// TwinCAT 3 PLC project Motors
// libraries:
//   Tc2_MC2, * (Beckhoff Automation GmbH)
//   Tc2_NC, * (Beckhoff Automation GmbH)
//   Tc2_Standard, * (Beckhoff Automation GmbH)
//   Tc2_System, * (Beckhoff Automation GmbH)
//   Tc3_Module, * (Beckhoff Automation GmbH)
// project tree:
//   Data types/ TComplexStruct.TcDUT, TSimpleStruct.TcDUT
//   Global Variables/ GVL_Axis1Ctrl.TcGVL, GVL_Axis2Ctrl.TcGVL, GVL_Axis3Ctrl.TcGVL, GVL_Axis4Ctrl.TcGVL, GVL_Axis5Ctrl.TcGVL, GVL_Axis6Ctrl.TcGVL, GVL_Brakes.TcGVL, GVL_NC.TcGVL, GVL_Remote.TcGVL
//   / GlobalTextList.TcGTLO, Standard.TcTTO, Visualization Manager.TcVMO (not stored)
//   POUs/ MAIN.TcPOU, POU_AbortMoves.TcPOU, POU_AxesError.TcPOU, POU_ClearAxesErrors.TcPOU, POU_Limits.TcPOU, POU_AxisMoveAbs.TcPOU, POU_Lights.TcPOU, POU_AxisClearError.TcPOU, POU_GetPosition.TcPOU, POUNCPowerOn.TcPOU, POU_AxisJogCtrl.TcPOU, POU_SetStatus.TcPOU
//   Visualizations/ Visualization.TcVIS
// real-time tasks:
//   TASK Motors: cycle T#10ms, priority 20, ADS port 350
// motion (NC):
//   TASK NC-Task 1 SAF: cycle T#2ms, priority 4, ADS port 501
//   TASK NC-Task 1 SVB: cycle T#10ms, priority 8, ADS port 511
//   AXIS Axis 1 (id 1)
//     Dynamic: AccelerationMaximum=50, DecelerationMaximum=50, Acceleration=0.5, Deceleration=0.5, Jerk=100
//     Velo: RefSearch=5, RefSync=5, SlowManual=0.5, FastManual=3, Fast=20, Maximum=20
//     PositionAreaControl: Range=0.00025
//     TargetPosControl: Range=0.00025, Time=0.5
//     OtherSettings: AllowMotionCmdToSlave=true, PulseDistancePos=0.5, PulseDistanceNeg=0.5
//     encoder EncType=29
//       EncPara: ScaleFactorNumerator=5e-05, Offset=-200, MaxCount=#xffffffff, ReferenceSystem=1
//         SoftEndMinControl: Enable=true, Range=-169
//         SoftEndMaxControl: Enable=true, Range=175
//         Inc: RefSoftSyncMask=#x0000ffff
//     drive DrvType=24
//       DrvPara: Inverse=true
//         Analog: VeloReferenz=15, VeloScale=0.5, ScaleFactorActTorque=0.1, AccOutputDelay=0.1
//         TimeComp: TaskDelayCycles=1
//     controller CtrType=3
//       CtrPara: PriorControlFactor=1
//         PosDiffControl: Range=1
//         PID: PosKp=5, DeadBandPosition=0.0002
//         Observer: BandWidth=20
//   AXIS Axis 2 (id 2)
//     Dynamic: AccelerationMaximum=50, DecelerationMaximum=50, Acceleration=1, Deceleration=1, Jerk=0.5
//     Velo: SlowManual=0.5, FastManual=5, Maximum=10
//     PositionAreaControl: Range=0.00025
//     TargetPosControl: Range=0.00025, Time=0.5
//     OtherSettings: AllowMotionCmdToSlave=true
//     encoder EncType=29
//       EncPara: ScaleFactorNumerator=5e-05, Offset=-130, MaxCount=#xffffffff, ReferenceSystem=1
//         SoftEndMinControl: Enable=true, Range=-71
//         SoftEndMaxControl: Enable=true, Range=69
//         Inc: RefSoftSyncMask=#x0000ffff
//     drive DrvType=24
//       DrvPara: Inverse=true
//         Analog: VeloReferenz=10, ScaleFactorActTorque=0.1
//         TimeComp: TaskDelayCycles=1
//     controller CtrType=3
//       CtrPara: PriorControlFactor=1
//         PosDiffControl: Range=1
//         PID: PosKp=100, DeadBandPosition=0.0002
//         Observer: BandWidth=20
//   AXIS Axis 3 (id 3)
//     Dynamic: AccelerationMaximum=50, DecelerationMaximum=50, Acceleration=0.5, Deceleration=0.5, Jerk=100
//     Velo: RefSearch=5, RefSync=5, SlowManual=0.5, FastManual=3, Maximum=20
//     PositionAreaControl: Range=0.00025
//     TargetPosControl: Range=0.00025, Time=0.5
//     OtherSettings: AllowMotionCmdToSlave=true
//     encoder EncType=29
//       EncPara: ScaleFactorNumerator=5e-05, Offset=-200, MaxCount=#xffffffff, ReferenceSystem=1
//         SoftEndMinControl: Enable=true, Range=-169
//         SoftEndMaxControl: Enable=true, Range=175
//         Inc: RefSoftSyncMask=#x0000ffff
//     drive DrvType=24
//       DrvPara: Inverse=true
//         Analog: VeloReferenz=15, ScaleFactorActTorque=0.1
//         TimeComp: TaskDelayCycles=1
//     controller CtrType=3
//       CtrPara: PriorControlFactor=1
//         PosDiffControl: Range=1
//         PID: PosKp=5
//         Observer: BandWidth=20
//   AXIS Axis 4 (id 4)
//     Dynamic: AccelerationMaximum=50, DecelerationMaximum=50, Acceleration=0.5, Deceleration=0.5, Jerk=0.5
//     Velo: RefSearch=5, RefSync=5, SlowManual=0.5, FastManual=3, Maximum=10
//     PositionAreaControl: Range=0.00025
//     TargetPosControl: Range=0.00025
//     OtherSettings: AllowMotionCmdToSlave=true
//     encoder EncType=29
//       EncPara: ScaleFactorNumerator=5e-05, Offset=-100, MaxCount=#xffffffff, ReferenceSystem=1
//         SoftEndMinControl: Enable=true, Range=-75
//         SoftEndMaxControl: Enable=true, Range=69
//         Inc: RefSoftSyncMask=#x0000ffff
//     drive DrvType=24
//       DrvPara: Inverse=true
//         Analog: VeloReferenz=10, ScaleFactorActTorque=0.1
//         TimeComp: TaskDelayCycles=1
//     controller CtrType=3
//       CtrPara: PriorControlFactor=1
//         PosDiffControl: Range=1
//         PID: PosKp=5, DeadBandPosition=0.0002
//         Observer: BandWidth=20
//   AXIS Axis 5 (id 5)
//     Dynamic: AccelerationMaximum=50, DecelerationMaximum=50, Acceleration=0.5, Deceleration=0.5, Jerk=100
//     Velo: RefSearch=5, RefSync=5, SlowManual=0.5, FastManual=3, Maximum=20
//     PositionAreaControl: Range=0.00025
//     TargetPosControl: Range=0.00025
//     OtherSettings: AllowMotionCmdToSlave=true
//     encoder EncType=29
//       EncPara: ScaleFactorNumerator=5e-05, Offset=-200, MaxCount=#xffffffff, ReferenceSystem=1
//         SoftEndMinControl: Enable=true, Range=-169
//         SoftEndMaxControl: Enable=true, Range=175
//         Inc: RefSoftSyncMask=#x0000ffff
//     drive DrvType=24
//       DrvPara: Inverse=true
//         Analog: VeloReferenz=15, ScaleFactorActTorque=0.1
//         TimeComp: TaskDelayCycles=1
//     controller CtrType=3
//       CtrPara: PriorControlFactor=1
//         PosDiffControl: Range=1
//         PID: PosKp=5
//         Observer: BandWidth=20
//   AXIS Axis 6 (id 6)
//     Dynamic: AccelerationMaximum=50, DecelerationMaximum=50, Acceleration=0.5, Deceleration=0.5, Jerk=0.5
//     Velo: RefSearch=5, RefSync=3, SlowManual=0.5, FastManual=3, Maximum=10
//     PositionAreaControl: Range=0.00025
//     TargetPosControl: Range=0.00025
//     OtherSettings: AllowMotionCmdToSlave=true
//     encoder EncType=29
//       EncPara: ScaleFactorNumerator=5e-05, Offset=-130, MaxCount=#xffffffff, ReferenceSystem=1
//         SoftEndMinControl: Enable=true, Range=-72
//         SoftEndMaxControl: Enable=true, Range=69
//         Inc: RefSoftSyncMask=#x0000ffff
//     drive DrvType=24
//       DrvPara: Inverse=true
//         Analog: VeloReferenz=10, ScaleFactorActTorque=0.1
//         TimeComp: TaskDelayCycles=1
//     controller CtrType=3
//       CtrPara: PriorControlFactor=1
//         PosDiffControl: Range=1
//         PID: PosKp=5, DeadBandPosition=0.0002
//         Observer: BandWidth=20
// I/O:
//   DEVICE Device 1 (EtherCAT), AmsNetId 5.68.208.232.2.1
//     Term 1 (EK1200) [EK1200-5000 EtherCAT Power supply (2A E-Bus)]
//       Term 2 (EL2008) [EL2008 8Ch. Dig. Output 24V, 0.5A]
//       Term 3 (EL9011) [EL9011 End Terminal]
//   DEVICE Device 4 (EtherCAT), AmsNetId 5.68.208.232.5.1
//     Term 4 (EK1914) [EK1914, 2 Ch. Safety Input/Output 24V,  TwinSAFE]
//       modules: Module 1 (FSOE), Module 2 (DIO)
//       Term 17 (EL9410) [EL9410 E-Bus Power Supplier  (Diagnostics)]
//       Term 5 (EL5042) [EL5042 2Ch. BiSS-C Encoder]
//       Term 6 (EL5042) [EL5042 2Ch. BiSS-C Encoder]
//       Term 7 (EL5042) [EL5042 2Ch. BiSS-C Encoder]
//       Term 8 (EL7041-0052) [EL7041-0052 1Ch. Stepper motor output stage (50V, 5A)]
//       Term 9 (EL7041-0052) [EL7041-0052 1Ch. Stepper motor output stage (50V, 5A)]
//       Term 10 (EL7041-0052) [EL7041-0052 1Ch. Stepper motor output stage (50V, 5A)]
//       Term 11 (EL7041-0052) [EL7041-0052 1Ch. Stepper motor output stage (50V, 5A)]
//       Term 12 (EL7041-0052) [EL7041-0052 1Ch. Stepper motor output stage (50V, 5A)]
//       Term 13 (EL7041-0052) [EL7041-0052 1Ch. Stepper motor output stage (50V, 5A)]
//       Term 11 (EL9011) [EL9011 End Terminal]
//   DEVICE Device 3 (RT-Ethernet Protocol) (disabled), AmsNetId 5.68.208.232.4.1
//   DEVICE Device 2 (USB) (disabled)
//     Box 1 (CX2100 Power Supply)
//   DEVICE Device 5 (NOV-DP-RAM) (disabled)
// variable links:
//   NC-Task 1 SAF/Axes/Axis 1 <-> Device 4 (EtherCAT)/Term 4 (EK1914)/Term 5 (EL5042)
//     Enc/Inputs/In/nComState @bit 1 <-> WcState/InputToggle
//     Enc/Inputs/In/nComState <-> WcState/WcState
//     Enc/Inputs/In/nDataIn1 <-> FB Inputs Channel 1/Position
//     Enc/Inputs/In/nState1 @bit 12 <-> FB Inputs Channel 1/Diag
//     Enc/Inputs/In/nState1 @bit 1 <-> FB Inputs Channel 1/Error
//     Enc/Inputs/In/nState1 @bit 14 <-> FB Inputs Channel 1/Input cycle counter
//     Enc/Inputs/In/nState1 @bit 2 <-> FB Inputs Channel 1/Ready
//     Enc/Inputs/In/nState1 @bit 13 <-> FB Inputs Channel 1/TxPDO State
//     Enc/Inputs/In/nState1 <-> FB Inputs Channel 1/Warning
//   NC-Task 1 SAF/Axes/Axis 1 <-> Device 4 (EtherCAT)/Term 4 (EK1914)/Term 8 (EL7041-0052)
//     Drive/Inputs/In/nState1 @bit 3 <-> STM Status/Error
//     Drive/Inputs/In/nState1 @bit 5 <-> STM Status/Moving negative
//     Drive/Inputs/In/nState1 @bit 4 <-> STM Status/Moving positive
//     Drive/Inputs/In/nState1 @bit 1 <-> STM Status/Ready
//     Drive/Inputs/In/nState1 <-> STM Status/Ready to enable
//     Drive/Inputs/In/nState1 @bit 6 <-> STM Status/Torque reduced
//     Drive/Inputs/In/nState1 @bit 2 <-> STM Status/Warning
//     Drive/Inputs/In/nState2 @bit 3 <-> STM Status/Digital input 1
//     Drive/Inputs/In/nState2 @bit 4 <-> STM Status/Digital input 2
//     Drive/Inputs/In/nState2 @bit 5 <-> STM Status/Sync error
//     Drive/Inputs/In/nState2 @bit 7 <-> STM Status/TxPDO Toggle
//     Drive/Inputs/In/nState4 @bit 1 <-> WcState/InputToggle
//     Drive/Inputs/In/nState4 <-> WcState/WcState
//     Drive/Outputs/Out/nCtrl1 <-> STM Control/Enable
//     Drive/Outputs/Out/nCtrl1 @bit 2 <-> STM Control/Reduce torque
//     Drive/Outputs/Out/nCtrl1 @bit 1 <-> STM Control/Reset
//     Drive/Outputs/Out/nDataOut2[0] <-> STM Velocity/Velocity
//   NC-Task 1 SAF/Axes/Axis 2 <-> Device 4 (EtherCAT)/Term 4 (EK1914)/Term 5 (EL5042)
//     Enc/Inputs/In/nComState @bit 1 <-> WcState/InputToggle
//     Enc/Inputs/In/nComState <-> WcState/WcState
//     Enc/Inputs/In/nDataIn1 <-> FB Inputs Channel 2/Position
//     Enc/Inputs/In/nState1 @bit 12 <-> FB Inputs Channel 2/Diag
//     Enc/Inputs/In/nState1 @bit 1 <-> FB Inputs Channel 2/Error
//     Enc/Inputs/In/nState1 @bit 14 <-> FB Inputs Channel 2/Input cycle counter
//     Enc/Inputs/In/nState1 @bit 2 <-> FB Inputs Channel 2/Ready
//     Enc/Inputs/In/nState1 @bit 13 <-> FB Inputs Channel 2/TxPDO State
//     Enc/Inputs/In/nState1 <-> FB Inputs Channel 2/Warning
//   NC-Task 1 SAF/Axes/Axis 2 <-> Device 4 (EtherCAT)/Term 4 (EK1914)/Term 9 (EL7041-0052)
//     Drive/Inputs/In/nState1 @bit 3 <-> STM Status/Status/Error
//     Drive/Inputs/In/nState1 @bit 5 <-> STM Status/Status/Moving negative
//     Drive/Inputs/In/nState1 @bit 4 <-> STM Status/Status/Moving positive
//     Drive/Inputs/In/nState1 @bit 1 <-> STM Status/Status/Ready
//     Drive/Inputs/In/nState1 <-> STM Status/Status/Ready to enable
//     Drive/Inputs/In/nState1 @bit 6 <-> STM Status/Status/Torque reduced
//     Drive/Inputs/In/nState1 @bit 2 <-> STM Status/Status/Warning
//     Drive/Inputs/In/nState2 @bit 5 <-> STM Status/Status/Sync error
//     Drive/Inputs/In/nState2 @bit 7 <-> STM Status/Status/TxPDO Toggle
//     Drive/Inputs/In/nState4 @bit 1 <-> WcState/InputToggle
//     Drive/Inputs/In/nState4 <-> WcState/WcState
//     Drive/Outputs/Out/nCtrl1 <-> STM Control/Control/Enable
//     Drive/Outputs/Out/nCtrl1 @bit 2 <-> STM Control/Control/Reduce torque
//     Drive/Outputs/Out/nCtrl1 @bit 1 <-> STM Control/Control/Reset
//     Drive/Outputs/Out/nDataOut2[0] <-> STM Velocity/Velocity
//   NC-Task 1 SAF/Axes/Axis 3 <-> Device 4 (EtherCAT)/Term 4 (EK1914)/Term 10 (EL7041-0052)
//     Drive/Inputs/In/nState1 @bit 3 <-> STM Status/Status/Error
//     Drive/Inputs/In/nState1 @bit 5 <-> STM Status/Status/Moving negative
//     Drive/Inputs/In/nState1 @bit 4 <-> STM Status/Status/Moving positive
//     Drive/Inputs/In/nState1 @bit 1 <-> STM Status/Status/Ready
//     Drive/Inputs/In/nState1 <-> STM Status/Status/Ready to enable
//     Drive/Inputs/In/nState1 @bit 6 <-> STM Status/Status/Torque reduced
//     Drive/Inputs/In/nState1 @bit 2 <-> STM Status/Status/Warning
//     Drive/Inputs/In/nState2 @bit 5 <-> STM Status/Status/Sync error
//     Drive/Inputs/In/nState2 @bit 7 <-> STM Status/Status/TxPDO Toggle
//     Drive/Inputs/In/nState4 @bit 1 <-> WcState/InputToggle
//     Drive/Inputs/In/nState4 <-> WcState/WcState
//     Drive/Outputs/Out/nCtrl1 <-> STM Control/Control/Enable
//     Drive/Outputs/Out/nCtrl1 @bit 2 <-> STM Control/Control/Reduce torque
//     Drive/Outputs/Out/nCtrl1 @bit 1 <-> STM Control/Control/Reset
//     Drive/Outputs/Out/nDataOut2[0] <-> STM Velocity/Velocity
//   NC-Task 1 SAF/Axes/Axis 3 <-> Device 4 (EtherCAT)/Term 4 (EK1914)/Term 6 (EL5042)
//     Enc/Inputs/In/nComState @bit 1 <-> WcState/InputToggle
//     Enc/Inputs/In/nComState <-> WcState/WcState
//     Enc/Inputs/In/nDataIn1 <-> FB Inputs Channel 1/Position
//     Enc/Inputs/In/nState1 @bit 12 <-> FB Inputs Channel 1/Status/Diag
//     Enc/Inputs/In/nState1 @bit 1 <-> FB Inputs Channel 1/Status/Error
//     Enc/Inputs/In/nState1 @bit 14 <-> FB Inputs Channel 1/Status/Input cycle counter
//     Enc/Inputs/In/nState1 @bit 2 <-> FB Inputs Channel 1/Status/Ready
//     Enc/Inputs/In/nState1 @bit 13 <-> FB Inputs Channel 1/Status/TxPDO State
//     Enc/Inputs/In/nState1 <-> FB Inputs Channel 1/Status/Warning
//   NC-Task 1 SAF/Axes/Axis 4 <-> Device 4 (EtherCAT)/Term 4 (EK1914)/Term 11 (EL7041-0052)
//     Drive/Inputs/In/nState1 @bit 3 <-> STM Status/Status/Error
//     Drive/Inputs/In/nState1 @bit 5 <-> STM Status/Status/Moving negative
//     Drive/Inputs/In/nState1 @bit 4 <-> STM Status/Status/Moving positive
//     Drive/Inputs/In/nState1 @bit 1 <-> STM Status/Status/Ready
//     Drive/Inputs/In/nState1 <-> STM Status/Status/Ready to enable
//     Drive/Inputs/In/nState1 @bit 6 <-> STM Status/Status/Torque reduced
//     Drive/Inputs/In/nState1 @bit 2 <-> STM Status/Status/Warning
//     Drive/Inputs/In/nState2 @bit 5 <-> STM Status/Status/Sync error
//     Drive/Inputs/In/nState2 @bit 7 <-> STM Status/Status/TxPDO Toggle
//     Drive/Inputs/In/nState4 @bit 1 <-> WcState/InputToggle
//     Drive/Inputs/In/nState4 <-> WcState/WcState
//     Drive/Outputs/Out/nCtrl1 <-> STM Control/Control/Enable
//     Drive/Outputs/Out/nCtrl1 @bit 2 <-> STM Control/Control/Reduce torque
//     Drive/Outputs/Out/nCtrl1 @bit 1 <-> STM Control/Control/Reset
//     Drive/Outputs/Out/nDataOut2[0] <-> STM Velocity/Velocity
//   NC-Task 1 SAF/Axes/Axis 4 <-> Device 4 (EtherCAT)/Term 4 (EK1914)/Term 6 (EL5042)
//     Enc/Inputs/In/nComState @bit 1 <-> WcState/InputToggle
//     Enc/Inputs/In/nComState <-> WcState/WcState
//     Enc/Inputs/In/nDataIn1 <-> FB Inputs Channel 2/Position
//     Enc/Inputs/In/nState1 @bit 12 <-> FB Inputs Channel 2/Status/Diag
//     Enc/Inputs/In/nState1 @bit 1 <-> FB Inputs Channel 2/Status/Error
//     Enc/Inputs/In/nState1 @bit 14 <-> FB Inputs Channel 2/Status/Input cycle counter
//     Enc/Inputs/In/nState1 @bit 2 <-> FB Inputs Channel 2/Status/Ready
//     Enc/Inputs/In/nState1 @bit 13 <-> FB Inputs Channel 2/Status/TxPDO State
//     Enc/Inputs/In/nState1 <-> FB Inputs Channel 2/Status/Warning
//   NC-Task 1 SAF/Axes/Axis 5 <-> Device 4 (EtherCAT)/Term 4 (EK1914)/Term 12 (EL7041-0052)
//     Drive/Inputs/In/nState1 @bit 3 <-> STM Status/Status/Error
//     Drive/Inputs/In/nState1 @bit 5 <-> STM Status/Status/Moving negative
//     Drive/Inputs/In/nState1 @bit 4 <-> STM Status/Status/Moving positive
//     Drive/Inputs/In/nState1 @bit 1 <-> STM Status/Status/Ready
//     Drive/Inputs/In/nState1 <-> STM Status/Status/Ready to enable
//     Drive/Inputs/In/nState1 @bit 6 <-> STM Status/Status/Torque reduced
//     Drive/Inputs/In/nState1 @bit 2 <-> STM Status/Status/Warning
//     Drive/Inputs/In/nState2 @bit 3 <-> STM Status/Status/Digital input 1
//     Drive/Inputs/In/nState2 @bit 4 <-> STM Status/Status/Digital input 2
//     Drive/Inputs/In/nState2 @bit 5 <-> STM Status/Status/Sync error
//     Drive/Inputs/In/nState2 @bit 7 <-> STM Status/Status/TxPDO Toggle
//     Drive/Inputs/In/nState4 @bit 1 <-> WcState/InputToggle
//     Drive/Inputs/In/nState4 <-> WcState/WcState
//     Drive/Outputs/Out/nCtrl1 <-> STM Control/Control/Enable
//     Drive/Outputs/Out/nCtrl1 @bit 2 <-> STM Control/Control/Reduce torque
//     Drive/Outputs/Out/nCtrl1 @bit 1 <-> STM Control/Control/Reset
//     Drive/Outputs/Out/nDataOut2[0] <-> STM Velocity/Velocity
//   NC-Task 1 SAF/Axes/Axis 5 <-> Device 4 (EtherCAT)/Term 4 (EK1914)/Term 7 (EL5042)
//     Enc/Inputs/In/nComState @bit 1 <-> WcState/InputToggle
//     Enc/Inputs/In/nComState <-> WcState/WcState
//     Enc/Inputs/In/nDataIn1 <-> FB Inputs Channel 1/Position
//     Enc/Inputs/In/nState1 @bit 12 <-> FB Inputs Channel 1/Status/Diag
//     Enc/Inputs/In/nState1 @bit 1 <-> FB Inputs Channel 1/Status/Error
//     Enc/Inputs/In/nState1 @bit 14 <-> FB Inputs Channel 1/Status/Input cycle counter
//     Enc/Inputs/In/nState1 @bit 2 <-> FB Inputs Channel 1/Status/Ready
//     Enc/Inputs/In/nState1 @bit 13 <-> FB Inputs Channel 1/Status/TxPDO State
//     Enc/Inputs/In/nState1 <-> FB Inputs Channel 1/Status/Warning
//   NC-Task 1 SAF/Axes/Axis 6 <-> Device 4 (EtherCAT)/Term 4 (EK1914)/Term 13 (EL7041-0052)
//     Drive/Inputs/In/nState1 @bit 3 <-> STM Status/Status/Error
//     Drive/Inputs/In/nState1 @bit 5 <-> STM Status/Status/Moving negative
//     Drive/Inputs/In/nState1 @bit 4 <-> STM Status/Status/Moving positive
//     Drive/Inputs/In/nState1 @bit 1 <-> STM Status/Status/Ready
//     Drive/Inputs/In/nState1 <-> STM Status/Status/Ready to enable
//     Drive/Inputs/In/nState1 @bit 6 <-> STM Status/Status/Torque reduced
//     Drive/Inputs/In/nState1 @bit 2 <-> STM Status/Status/Warning
//     Drive/Inputs/In/nState2 @bit 5 <-> STM Status/Status/Sync error
//     Drive/Inputs/In/nState2 @bit 7 <-> STM Status/Status/TxPDO Toggle
//     Drive/Inputs/In/nState4 @bit 1 <-> WcState/InputToggle
//     Drive/Inputs/In/nState4 <-> WcState/WcState
//     Drive/Outputs/Out/nCtrl1 <-> STM Control/Control/Enable
//     Drive/Outputs/Out/nCtrl1 @bit 2 <-> STM Control/Control/Reduce torque
//     Drive/Outputs/Out/nCtrl1 @bit 1 <-> STM Control/Control/Reset
//     Drive/Outputs/Out/nDataOut2[0] <-> STM Velocity/Velocity
//   NC-Task 1 SAF/Axes/Axis 6 <-> Device 4 (EtherCAT)/Term 4 (EK1914)/Term 7 (EL5042)
//     Enc/Inputs/In/nComState @bit 1 <-> WcState/InputToggle
//     Enc/Inputs/In/nComState <-> WcState/WcState
//     Enc/Inputs/In/nDataIn1 <-> FB Inputs Channel 2/Position
//     Enc/Inputs/In/nState1 @bit 12 <-> FB Inputs Channel 2/Status/Diag
//     Enc/Inputs/In/nState1 @bit 1 <-> FB Inputs Channel 2/Status/Error
//     Enc/Inputs/In/nState1 @bit 14 <-> FB Inputs Channel 2/Status/Input cycle counter
//     Enc/Inputs/In/nState1 @bit 2 <-> FB Inputs Channel 2/Status/Ready
//     Enc/Inputs/In/nState1 @bit 13 <-> FB Inputs Channel 2/Status/TxPDO State
//     Enc/Inputs/In/nState1 <-> FB Inputs Channel 2/Status/Warning
//   Motors/Motors Instance <-> Device 1 (EtherCAT)/Term 1 (EK1200)/Term 2 (EL2008)
//     Standard Outputs/MAIN.bAxis{1..6}Brake <-> Channel {1..6}/Output  (6 links)
//   Motors/Motors Instance <-> Device 4 (EtherCAT)/Term 4 (EK1914)
//     Standard Inputs/MAIN.bESTOP <-> Module 2 (DIO)/DIO Inputs/Input 0
//     Standard Outputs/POU_Lights.bLightAmber <-> Module 2 (DIO)/DIO Outputs/Output 1
//     Standard Outputs/POU_Lights.bLightGreen <-> Module 2 (DIO)/DIO Outputs/Output 0
//     Standard Outputs/POU_Lights.bLightRed <-> Module 2 (DIO)/DIO Outputs/Output 2
//   Motors/Motors Instance <-> Device 4 (EtherCAT)/Term 4 (EK1914)/Term 10 (EL7041-0052)
//     Standard Inputs/POUNCPowerOn.bAxis3LimitNegI <-> STM Status/Status/Digital input 2
//     Standard Inputs/POUNCPowerOn.bAxis3LimitPosI <-> STM Status/Status/Digital input 1
//     Standard Inputs/POU_Limits.bAxis3LimitNegI <-> STM Status/Status/Digital input 2
//     Standard Inputs/POU_Limits.bAxis3LimitPosI <-> STM Status/Status/Digital input 1
//   Motors/Motors Instance <-> Device 4 (EtherCAT)/Term 4 (EK1914)/Term 11 (EL7041-0052)
//     Standard Inputs/POUNCPowerOn.bAxis4LimitNegI <-> STM Status/Status/Digital input 2
//     Standard Inputs/POUNCPowerOn.bAxis4LimitPosI <-> STM Status/Status/Digital input 1
//     Standard Inputs/POU_Limits.bAxis4LimitNegI <-> STM Status/Status/Digital input 2
//     Standard Inputs/POU_Limits.bAxis4LimitPosI <-> STM Status/Status/Digital input 1
//   Motors/Motors Instance <-> Device 4 (EtherCAT)/Term 4 (EK1914)/Term 12 (EL7041-0052)
//     Standard Inputs/POUNCPowerOn.bAxis5LimitNegI <-> STM Status/Status/Digital input 2
//     Standard Inputs/POUNCPowerOn.bAxis5LimitPosI <-> STM Status/Status/Digital input 1
//     Standard Inputs/POU_Limits.bAxis5LimitNegI <-> STM Status/Status/Digital input 2
//     Standard Inputs/POU_Limits.bAxis5LimitPosI <-> STM Status/Status/Digital input 1
//   Motors/Motors Instance <-> Device 4 (EtherCAT)/Term 4 (EK1914)/Term 13 (EL7041-0052)
//     Standard Inputs/POUNCPowerOn.bAxis6LimitNegI <-> STM Status/Status/Digital input 2
//     Standard Inputs/POUNCPowerOn.bAxis6LimitPosI <-> STM Status/Status/Digital input 1
//     Standard Inputs/POU_Limits.bAxis6LimitNegI <-> STM Status/Status/Digital input 2
//     Standard Inputs/POU_Limits.bAxis6LimitPosI <-> STM Status/Status/Digital input 1
//   Motors/Motors Instance <-> Device 4 (EtherCAT)/Term 4 (EK1914)/Term 8 (EL7041-0052)
//     Standard Inputs/POUNCPowerOn.bAxis1LimitNegI <-> STM Status/Digital input 2
//     Standard Inputs/POUNCPowerOn.bAxis1LimitPosI <-> STM Status/Digital input 1
//     Standard Inputs/POU_Limits.bAxis1LimitNegI <-> STM Status/Digital input 2
//     Standard Inputs/POU_Limits.bAxis1LimitPosI <-> STM Status/Digital input 1
//   Motors/Motors Instance <-> Device 4 (EtherCAT)/Term 4 (EK1914)/Term 9 (EL7041-0052)
//     Standard Inputs/POUNCPowerOn.bAxis2LimitNegI <-> STM Status/Status/Digital input 2
//     Standard Inputs/POUNCPowerOn.bAxis2LimitPosI <-> STM Status/Status/Digital input 1
//     Standard Inputs/POU_Limits.bAxis2LimitNegI <-> STM Status/Status/Digital input 2
//     Standard Inputs/POU_Limits.bAxis2LimitPosI <-> STM Status/Status/Digital input 1
//   Motors/Motors Instance <-> NC-Task 1 SAF/Axes/Axis 1
//     Standard Inputs/GVL_NC.Axis1.NcToPlc <-> Outputs/ToPlc
//     Standard Inputs/POU_AxesError.bAxis1ErrorI <-> Outputs/ToPlc/StateDWord/Error
//     Standard Outputs/GVL_NC.Axis1.PlcToNc <-> Inputs/FromPlc
//   Motors/Motors Instance <-> NC-Task 1 SAF/Axes/Axis 2
//     Standard Inputs/GVL_NC.Axis2.NcToPlc <-> Outputs/ToPlc
//     Standard Inputs/POU_AxesError.bAxis2ErrorI <-> Outputs/ToPlc/StateDWord/Error
//     Standard Outputs/GVL_NC.Axis2.PlcToNc <-> Inputs/FromPlc
//   Motors/Motors Instance <-> NC-Task 1 SAF/Axes/Axis 3
//     Standard Inputs/GVL_NC.Axis3.NcToPlc <-> Outputs/ToPlc
//     Standard Inputs/POU_AxesError.bAxis3ErrorI <-> Outputs/ToPlc/StateDWord/Error
//     Standard Outputs/GVL_NC.Axis3.PlcToNc <-> Inputs/FromPlc
//   Motors/Motors Instance <-> NC-Task 1 SAF/Axes/Axis 4
//     Standard Inputs/GVL_NC.Axis4.NcToPlc <-> Outputs/ToPlc
//     Standard Inputs/POU_AxesError.bAxis4ErrorI <-> Outputs/ToPlc/StateDWord/Error
//     Standard Outputs/GVL_NC.Axis4.PlcToNc <-> Inputs/FromPlc
//   Motors/Motors Instance <-> NC-Task 1 SAF/Axes/Axis 5
//     Standard Inputs/GVL_NC.Axis5.NcToPlc <-> Outputs/ToPlc
//     Standard Inputs/POU_AxesError.bAxis5ErrorI <-> Outputs/ToPlc/StateDWord/Error
//     Standard Outputs/GVL_NC.Axis5.PlcToNc <-> Inputs/FromPlc
//   Motors/Motors Instance <-> NC-Task 1 SAF/Axes/Axis 6
//     Standard Inputs/GVL_NC.Axis6.NcToPlc <-> Outputs/ToPlc
//     Standard Inputs/POU_AxesError.bAxis6ErrorI <-> Outputs/ToPlc/StateDWord/Error
//     Standard Outputs/GVL_NC.Axis6.PlcToNc <-> Inputs/FromPlc

CONFIGURATION Motors
    RESOURCE PLC ON TwinCAT3
        TASK Standard(INTERVAL := T#10ms, PRIORITY := 20);
        PROGRAM MAIN WITH Standard : MAIN;
    END_RESOURCE
END_CONFIGURATION

// ---- Data types/TComplexStruct.TcDUT
TYPE TComplexStruct :
STRUCT
	intVal : INT:=1200;
	dintArr: ARRAY[0..3] OF DINT:=[ 1,2,3,4];
	boolVal: BOOL := FALSE;
	byteVal: BYTE:=10;
	stringVal : STRING(5) := 'hallo';
	simpleStruct1: TSimpleStruct;
END_STRUCT
END_TYPE

// ---- Data types/TSimpleStruct.TcDUT
TYPE TSimpleStruct :
STRUCT
	lrealVal: LREAL := 1.23;
	dintVal1: DINT := 120000;
END_STRUCT
END_TYPE

// ---- Global Variables/GVL_Axis1Ctrl.TcGVL
VAR_GLOBAL
	bAxis1Enable:BOOL;
	bAxis1EnablePos:BOOL:=TRUE;
	bAxis1EnableNeg:BOOL:=TRUE;
	bAxis1JogPos:BOOL;
	bAxis1JogNeg:BOOL;
	rAxis1Target:LREAL;
	bAxis1MoveABS:BOOL;
	rAxis1Vel:REAL;
	bAxis1PosLimit:BOOL:=TRUE;
	bAxis1NegLimit:BOOL:=TRUE;
	bAxis1GetPos:BOOL:=FALSE;
	rAxis1Position:LREAL;
	bAxis1InPosition:BOOL;
	iAxis1Error:UDINT;
	bAxis1Error:BOOL;
	bReset1Done:BOOL:=FALSE;
	
	
	
END_VAR

// ---- Global Variables/GVL_Axis2Ctrl.TcGVL
VAR_GLOBAL
	bAxis2Enable:BOOL;
	bAxis2EnablePos:BOOL:=TRUE;
	bAxis2EnableNeg:BOOL:=TRUE;
	bAxis2JogPos:BOOL;
	bAxis2JogNeg:BOOL;
	rAxis2Target:LREAL;
	bAxis2MoveABS:BOOL;
	rAxis2Vel:REAL;
	bAxis2PosLimit:BOOL:=TRUE;
	bAxis2NegLimit:BOOL:=TRUE;
	bAxis2GetPos:BOOL:=FALSE;
	rAxis2Position:LREAL;
	bAxis2InPosition:BOOL;
	iAxis2Error:UDINT;
	bAxis2Error:BOOL;
	bReset2Done:BOOL:=FALSE;
END_VAR

// ---- Global Variables/GVL_Axis3Ctrl.TcGVL
VAR_GLOBAL
	bAxis3Enable:BOOL;
	bAxis3EnablePos:BOOL:=TRUE;
	bAxis3EnableNeg:BOOL:=TRUE;
	bAxis3JogPos:BOOL;
	bAxis3JogNeg:BOOL;
	rAxis3Target:LREAL;
	bAxis3MoveABS:BOOL;
	rAxis3Vel:REAL;
	bAxis3PosLimit:BOOL:=TRUE;
	bAxis3NegLimit:BOOL:=TRUE;
	bAxis3GetPos:BOOL:=FALSE;
	rAxis3Position:LREAL;
	bAxis3InPosition:BOOL;
	iAxis3Error:UDINT;
	bAxis3Error:BOOL;
	bReset3Done:BOOL:=FALSE;
END_VAR

// ---- Global Variables/GVL_Axis4Ctrl.TcGVL
VAR_GLOBAL
	bAxis4Enable:BOOL;
	bAxis4EnablePos:BOOL:=TRUE;
	bAxis4EnableNeg:BOOL:=TRUE;
	bAxis4JogPos:BOOL;
	bAxis4JogNeg:BOOL;
	rAxis4Target:LREAL;
	bAxis4MoveABS:BOOL;
	rAxis4Vel:REAL;
	bAxis4PosLimit:BOOL:=TRUE;
	bAxis4NegLimit:BOOL:=TRUE;
	bAxis4GetPos:BOOL:=FALSE;
	rAxis4Position:LREAL;
	bAxis4InPosition:BOOL;
	iAxis4Error:UDINT;
	bAxis4Error:BOOL;
	bReset4Done:BOOL:=FALSE;
END_VAR

// ---- Global Variables/GVL_Axis5Ctrl.TcGVL
VAR_GLOBAL
	bAxis5Enable:BOOL;
	bAxis5EnablePos:BOOL:=TRUE;
	bAxis5EnableNeg:BOOL:=TRUE;
	bAxis5JogPos:BOOL;
	bAxis5JogNeg:BOOL;
	rAxis5Target:LREAL;
	bAxis5MoveABS:BOOL;
	rAxis5Vel:REAL;
	bAxis5PosLimit:BOOL:=TRUE;
	bAxis5NegLimit:BOOL:=TRUE;
	bAxis5GetPos:BOOL:=FALSE;
	rAxis5Position:LREAL;
	bAxis5InPosition:BOOL;	
	iAxis5Error:UDINT;
	bAxis5Error:BOOL;
	bReset5Done:BOOL:=FALSE;
END_VAR

// ---- Global Variables/GVL_Axis6Ctrl.TcGVL
VAR_GLOBAL
	bAxis6Enable:BOOL;
	bAxis6EnablePos:BOOL:=TRUE;
	bAxis6EnableNeg:BOOL:=TRUE;
	bAxis6JogPos:BOOL;
	bAxis6JogNeg:BOOL;
	rAxis6Target:LREAL;
	bAxis6MoveABS:BOOL;
	rAxis6Vel:REAL;
	bAxis6PosLimit:BOOL:=TRUE;
	bAxis6NegLimit:BOOL:=TRUE;
	bAxis6GetPos:BOOL:=FALSE;
	rAxis6Position:LREAL;
	bAxis6InPosition:BOOL;
	iAxis6Error:UDINT;
	bAxis6Error:BOOL;
	bReset6Done:BOOL:=FALSE;
END_VAR

// ---- Global Variables/GVL_Brakes.TcGVL
VAR_GLOBAL
	bAxis1Brake:BOOL;
	bAxis2Brake:BOOL;
	bAxis3Brake:BOOL;
	bAxis4Brake:BOOL;
	bAxis5Brake:BOOL;
	bAxis6Brake:BOOL;
END_VAR

// ---- Global Variables/GVL_NC.TcGVL
VAR_GLOBAL
	Axis1:AXIS_REF;
	stAxis1:ST_AxisStatus;
	Axis2:AXIS_REF;
	stAxis2:ST_AxisStatus;
	Axis3:AXIS_REF;
	stAxis3:ST_AxisStatus;
	Axis4:AXIS_REF;
	stAxis4:ST_AxisStatus;	
	Axis5:AXIS_REF;
	stAxis5:ST_AxisStatus;
	Axis6:AXIS_REF;
	stAxis6:ST_AxisStatus;
	rAxisVelV:REAL:=2;
	rAxisVelH:REAL:=2;
	bLimits:BOOL;
	bMotorError:BOOL:=FALSE;
	bReSetMotor:BOOL:=FALSE;
	bAbortMove:BOOL:=FALSE;
END_VAR

// ---- Global Variables/GVL_Remote.TcGVL
VAR_GLOBAL
	bRemote:BOOL:=TRUE;
END_VAR

// ---- POUs/MAIN.TcPOU
PROGRAM MAIN
VAR
	(*primitive Types*)
	Bool1:BOOL := FALSE;
	int1:INT :=0;
	dint1:DINT:=125000;
	usint1:USINT:=200;
	real1:REAL:= 1.2;
	lreal1:LREAL:=3.5;
	rConst:REAL;
	bClearAxesErrorm:BOOL:=FALSE;
	
	bAxis1Brake  AT%Q* : BOOL;
	bAxis2Brake  AT%Q* : BOOL;
	bAxis3Brake  AT%Q* : BOOL;
	bAxis4Brake  AT%Q* : BOOL;
	bAxis5Brake  AT%Q* : BOOL;
	bAxis6Brake  AT%Q* : BOOL;
	
	
	
	(*string Types*)
	str1:STRING := 'this is a test string';
	str2:STRING(5) := 'hallo';
	
	(*struct Types*)
	complexStruct1 : TComplexStruct;

	bESTOP AT%I* :BOOL;
	i: INT;
//Axis 1 Var	
	fbReadAxis1Status:MC_ReadStatus;
	bAxesEnablem:BOOL:=FALSE;
	bAxis1JogPosm:BOOL:=FALSE;
	bAxis1JogNegm:BOOL:=FALSE;
	rAxis1Targetm:LREAL:=0;
	rAxis1Positionm:LREAL:=0;
	bAxis1LimitPos:BOOL;
	bAxis1LimitNeg:BOOL;
	bAxis1MoveABSm:BOOL:=FALSE;
	bAxis1GetPosm:BOOL:=FALSE;
	bAxis1InPositionm:BOOL;
//Axis 2 Var	
	fbReadAxis2Status:MC_ReadStatus;
	bAxis2Enablem:BOOL:=FALSE;
	bAxis2JogPosm:BOOL:=FALSE;
	bAxis2JogNegm:BOOL:=FALSE;
	rAxis2Targetm:LREAL:=0;
	rAxis2Positionm:LREAL:=0;
	bAxis2LimitPos:BOOL;
	bAxis2LimitNeg:BOOL;
	bAxis2MoveABSm:BOOL:=FALSE;
	bAxis2InPositionm:BOOL;
//Axis 3 Var	
	fbReadAxis3Status:MC_ReadStatus;	
	bAxis3Enablem:BOOL:=FALSE;
	bAxis3JogPosm:BOOL:=FALSE;
	bAxis3JogNegm:BOOL:=FALSE;
	rAxis3Targetm:LREAL:=0;
	rAxis3Positionm:LREAL:=0;
	bAxis3LimitPos:BOOL;
	bAxis3LimitNeg:BOOL;
	bAxis3MoveABSm:BOOL:=FALSE;
	bAxis3InPositionm:BOOL;
//Axis 4 Var	
	fbReadAxis4Status:MC_ReadStatus;
	bAxis4JogPosm:BOOL:=FALSE;
	bAxis4JogNegm:BOOL:=FALSE;
	rAxis4Targetm:LREAL:=0;
	rAxis4Positionm:LREAL:=0;
	bAxis4LimitPos:BOOL;
	bAxis4LimitNeg:BOOL;
	bAxis4MoveABSm:BOOL:=FALSE;
	bAxis4InPositionm:BOOL;
//Axis 5 Var	
	fbReadAxis5Status:MC_ReadStatus;
	bAxis5JogPosm:BOOL:=FALSE;
	bAxis5JogNegm:BOOL:=FALSE;
	rAxis5Targetm:LREAL:=0;
	rAxis5Positionm:LREAL:=0;
	bAxis5LimitPos:BOOL;
	bAxis5LimitNeg:BOOL;
	bAxis5MoveABSm:BOOL:=FALSE;
	bAxis5InPositionm:BOOL;
//Axis 6 Var	
	fbReadAxis6Status:MC_ReadStatus;
	bAxis6JogPosm:BOOL:=FALSE;
	bAxis6JogNegm:BOOL:=FALSE;
	rAxis6Targetm:LREAL:=0;
	rAxis6Positionm:LREAL:=0;
	bAxis6LimitPos:BOOL;
	bAxis6LimitNeg:BOOL;
	bAxis6MoveABSm:BOOL:=FALSE;
	bAxis6InPositionm:BOOL;

	fbMoveAbs: MC_MoveAbsolute;
	fbMoveAbs2: MC_MoveAbsolute;
END_VAR


	POU_GetPosition();
	POU_Lights(bEStop:=bEStop);
	POU_Limits();
	POU_AxesError();
IF bESTOP AND bLimits AND bMotorError
	THEN
	IF bRemote 
	THEN

	//Axis 1
	bAxis1Enable:=bAxesEnablem;
	bAxis1Brake:=bAxis1Enable;
	rAxis1Target:=rAxis1Targetm;
	bAxis1MoveABS:=bAxis1MoveABSm;
	rAxis1Positionm:=rAxis1Position;
	bAxis1InPositionm:=bAxis1InPosition;

	//Axis 2
	bAxis2Enable:=bAxesEnablem;
	bAxis2Brake:=bAxis2Enable;
	rAxis2Target:=rAxis2Targetm;
	bAxis2MoveABS:=bAxis2MoveABSm;
	rAxis2Positionm:=rAxis2Position;
	bAxis2InPositionm:=bAxis2InPosition;

	//Axis 3
	bAxis3Enable:=bAxesEnablem;
	bAxis3Brake:=bAxis3Enable;
	rAxis3Target:=rAxis3Targetm;
	bAxis3MoveABS:=bAxis3MoveABSm;
	rAxis3Positionm:=rAxis3Position;
	bAxis3InPositionm:=bAxis3InPosition;

	//Axis 4
	bAxis4Enable:=bAxesEnablem;
	bAxis4Brake:=bAxis4Enable;
	rAxis4Target:=rAxis4Targetm;
	bAxis4MoveABS:=bAxis4MoveABSm;
	rAxis4Positionm:=rAxis4Position;
	bAxis4InPositionm:=bAxis4InPosition;

	//Axis 5
	bAxis5Enable:=bAxesEnablem;
	bAxis5Brake:=bAxis5Enable;
	rAxis5Target:=rAxis5Targetm;
	bAxis5MoveABS:=bAxis5MoveABSm;
	rAxis5Positionm:=rAxis5Position;
	bAxis5InPositionm:=bAxis5InPosition;

	//Axis 6
	bAxis6Enable:=bAxesEnablem;
	bAxis6Brake:=bAxis6Enable;
	rAxis6Target:=rAxis6Targetm;
	bAxis6MoveABS:=bAxis6MoveABSm;
	rAxis6Positionm:=rAxis6Position;
	bAxis6InPositionm:=bAxis6InPosition;

	POUNCPowerOn();
	POU_AxisJogCtrl();
	POU_AxisMoveABS();

	END_IF;
ELSE
	bAxis1Enable:=FALSE;
	bAxis2Enable:=FALSE;
	bAxis3Enable:=FALSE;
	bAxis4Enable:=FALSE;
	bAxis5Enable:=FALSE;
	bAxis6Enable:=FALSE;
	bAxis1MoveABS:=FALSE;
	bAxis2MoveABS:=FALSE;
	bAxis3MoveABS:=FALSE;
	bAxis4MoveABS:=FALSE;
	bAxis5MoveABS:=FALSE;
	bAxis6MoveABS:=FALSE;
	bAxis1Brake:=FALSE;
	bAxis2Brake:=FALSE;
	bAxis3Brake:=FALSE;
	bAxis4Brake:=FALSE;
	bAxis5Brake:=FALSE;
	bAxis6Brake:=FALSE;
	//needs to set move abs execute to false both 1 and 2
	POUNCPowerOn();
END_IF;
IF bClearAxesErrorm
	THEN
	int1:=int1+1;
	bReSetMotor:=TRUE;
	POU_ClearAxesErrors();

	IF bReset2Done
		THEN
			bReSetMotor:=FALSE;
			POU_ClearAxesErrors();
			bClearAxesErrorm:=FALSE;
	END_IF

END_IF

END_PROGRAM

// ---- POUs/POU_GetPosition.TcPOU
PROGRAM POU_GetPosition
VAR
	fb_Axis1Position:MC_ReadActualPosition;
	fb_Axis2Position:MC_ReadActualPosition;
	fb_Axis3Position:MC_ReadActualPosition;
	fb_Axis4Position:MC_ReadActualPosition;
	fb_Axis5Position:MC_ReadActualPosition;
	fb_Axis6Position:MC_ReadActualPosition;
END_VAR

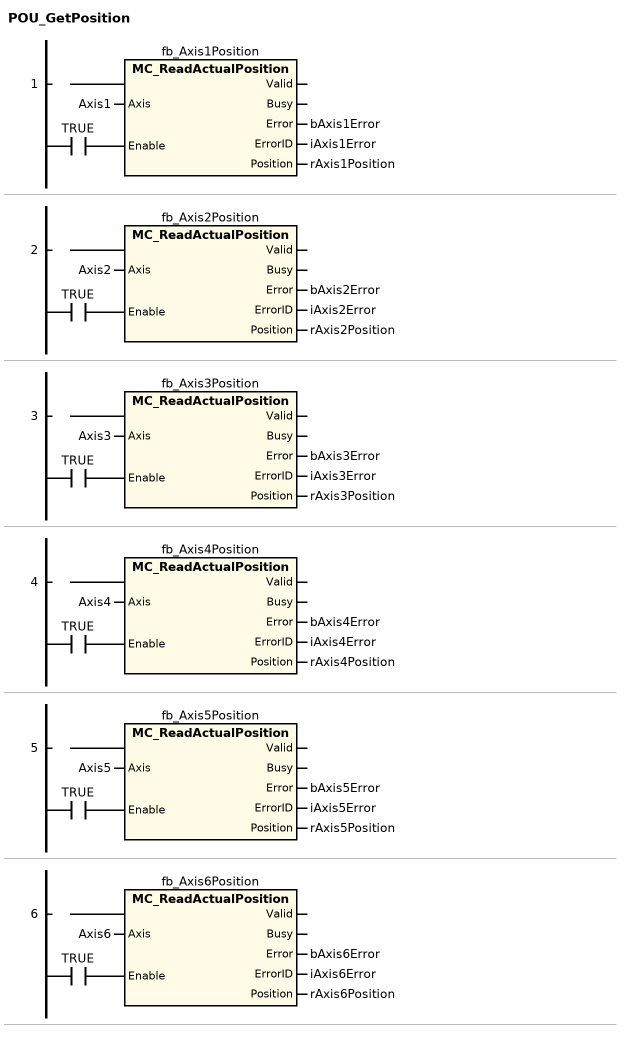
// NETWORK 1
fb_Axis1Position(
    Axis := Axis1,
    Enable := TRUE,
    Error => bAxis1Error,
    ErrorID => iAxis1Error,
    Position => rAxis1Position); // MC_ReadActualPosition

// NETWORK 2
fb_Axis2Position(
    Axis := Axis2,
    Enable := TRUE,
    Error => bAxis2Error,
    ErrorID => iAxis2Error,
    Position => rAxis2Position); // MC_ReadActualPosition

// NETWORK 3
fb_Axis3Position(
    Axis := Axis3,
    Enable := TRUE,
    Error => bAxis3Error,
    ErrorID => iAxis3Error,
    Position => rAxis3Position); // MC_ReadActualPosition

// NETWORK 4
fb_Axis4Position(
    Axis := Axis4,
    Enable := TRUE,
    Error => bAxis4Error,
    ErrorID => iAxis4Error,
    Position => rAxis4Position); // MC_ReadActualPosition

// NETWORK 5
fb_Axis5Position(
    Axis := Axis5,
    Enable := TRUE,
    Error => bAxis5Error,
    ErrorID => iAxis5Error,
    Position => rAxis5Position); // MC_ReadActualPosition

// NETWORK 6
fb_Axis6Position(
    Axis := Axis6,
    Enable := TRUE,
    Error => bAxis6Error,
    ErrorID => iAxis6Error,
    Position => rAxis6Position); // MC_ReadActualPosition

END_PROGRAM

// ---- POUs/POU_Lights.TcPOU
PROGRAM POU_Lights
VAR_INPUT
bAxesEnablem:BOOL;
bEStop:BOOL;
END_VAR
VAR
tTimeLightOn:TIME:=T#0S;
tTimeStartMove:TIME;
tCurrentLight:TIME;
tCurrentMoveDur:TIME;
bLightRed  AT%Q* : BOOL;
bLightAmber  AT%Q* : BOOL;
bLightGreen  AT%Q* : BOOL;
END_VAR

IF bEStop AND bLimits AND bMotorError
	THEN
	

IF bAxis1Enable OR bAxis2Enable OR bAxis3Enable OR bAxis4Enable OR bAxis5Enable OR bAxis6Enable
	
	THEN
	tCurrentLight:=TIME();
	tCurrentMoveDur:=tCurrentLight-tTimeLightOn;
	IF (tCurrentMoveDur < T#1S)  
		THEN
		bLightRed:=FALSE;
		bLightAmber:=TRUE;
		bLightGreen:=FALSE;
	END_IF
	IF (tCurrentMoveDur > T#1S)AND (tCurrentMoveDur < T#2S)
		THEN
		bLightRed:=FALSE;
		bLightAmber:=FALSE;
		bLightGreen:=FALSE;
	END_IF
	IF (tCurrentMoveDur > T#2S)
		THEN
		tTimeLightOn:=TIME();
	END_IF
	ELSE
	tTimeLightOn:=TIME();	
	bLightRed:=FALSE;
	bLightAmber:=FALSE;
	bLightGreen:=TRUE;
END_IF
ELSE
	bLightRed:=TRUE;
	bLightAmber:=FALSE;
	bLightGreen:=FALSE;
END_IF

END_PROGRAM

// ---- POUs/POU_Limits.TcPOU
PROGRAM POU_Limits
VAR
	bAxis1LimitPosI AT%I* :BOOL;
	bAxis1LimitNegI AT%I* :BOOL;
	bAxis2LimitPosI AT%I* :BOOL;
	bAxis2LimitNegI AT%I* :BOOL;
	bAxis3LimitPosI AT%I* :BOOL;
	bAxis3LimitNegI AT%I* :BOOL;
	bAxis4LimitPosI AT%I* :BOOL;
	bAxis4LimitNegI AT%I* :BOOL;
	bAxis5LimitPosI AT%I* :BOOL;
	bAxis5LimitNegI AT%I* :BOOL;
	bAxis6LimitPosI AT%I* :BOOL;
	bAxis6LimitNegI AT%I* :BOOL;
END_VAR

IF bAxis1LimitPosI AND bAxis1LimitNegI AND bAxis2LimitPosI AND bAxis2LimitNegI AND bAxis3LimitPosI AND bAxis3LimitNegI AND bAxis4LimitPosI AND bAxis4LimitNegI AND bAxis5LimitPosI AND bAxis5LimitNegI AND bAxis6LimitPosI AND bAxis6LimitNegI
	THEN bLimits:= TRUE;
	ELSE bLimits:=FALSE;
END_IF

END_PROGRAM

// ---- POUs/POU_AxesError.TcPOU
PROGRAM POU_AxesError
VAR
	bAxis1ErrorI AT%I* :BOOL;
	bAxis2ErrorI AT%I* :BOOL;
	bAxis3ErrorI AT%I* :BOOL;
	bAxis4ErrorI AT%I* :BOOL;
	bAxis5ErrorI AT%I* :BOOL;
	bAxis6ErrorI AT%I* :BOOL;
END_VAR

IF bAxis1ErrorI OR bAxis2ErrorI OR bAxis3ErrorI OR bAxis4ErrorI OR bAxis5ErrorI OR bAxis6ErrorI
	THEN
	bMotorError:=FALSE;
	ELSE
		bMotorError:=TRUE;
END_IF

END_PROGRAM

// ---- POUs/POUNCPowerOn.TcPOU
PROGRAM POUNCPowerOn
VAR
	fbAxis1PowerOn:MC_Power;
	fbAxis2PowerOn:MC_Power;
	fbAxis3PowerOn:MC_Power;
	fbAxis4PowerOn:MC_Power;
	fbAxis5PowerOn:MC_Power;
	fbAxis6PowerOn:MC_Power;
	bAxis1LimitPosI AT%I* :BOOL;
	bAxis1LimitNegI AT%I* :BOOL;
	bAxis2LimitPosI AT%I* :BOOL;
	bAxis2LimitNegI AT%I* :BOOL;
	bAxis3LimitPosI AT%I* :BOOL;
	bAxis3LimitNegI AT%I* :BOOL;
	bAxis4LimitPosI AT%I* :BOOL;
	bAxis4LimitNegI AT%I* :BOOL;
	bAxis5LimitPosI AT%I* :BOOL;
	bAxis5LimitNegI AT%I* :BOOL;
	bAxis6LimitPosI AT%I* :BOOL;
	bAxis6LimitNegI AT%I* :BOOL;
END_VAR

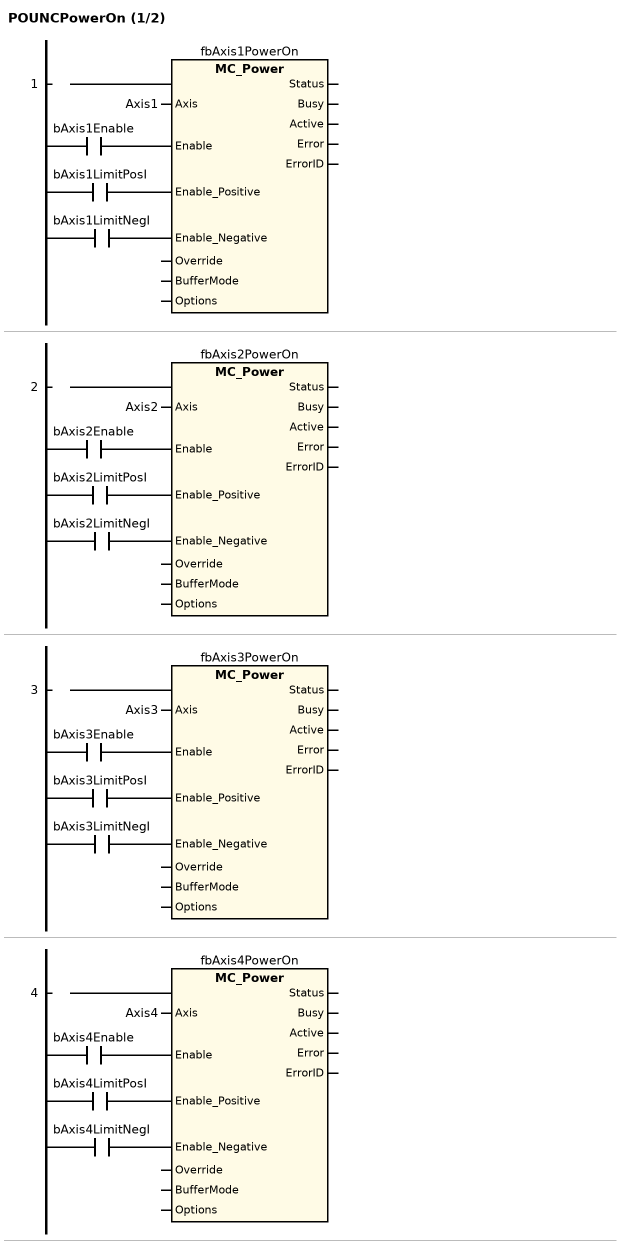
// NETWORK 1
fbAxis1PowerOn(
    Axis := Axis1,
    Enable := bAxis1Enable,
    Enable_Positive := bAxis1LimitPosI,
    Enable_Negative := bAxis1LimitNegI); // MC_Power

// NETWORK 2
fbAxis2PowerOn(
    Axis := Axis2,
    Enable := bAxis2Enable,
    Enable_Positive := bAxis2LimitPosI,
    Enable_Negative := bAxis2LimitNegI); // MC_Power

// NETWORK 3
fbAxis3PowerOn(
    Axis := Axis3,
    Enable := bAxis3Enable,
    Enable_Positive := bAxis3LimitPosI,
    Enable_Negative := bAxis3LimitNegI); // MC_Power

// NETWORK 4
fbAxis4PowerOn(
    Axis := Axis4,
    Enable := bAxis4Enable,
    Enable_Positive := bAxis4LimitPosI,
    Enable_Negative := bAxis4LimitNegI); // MC_Power

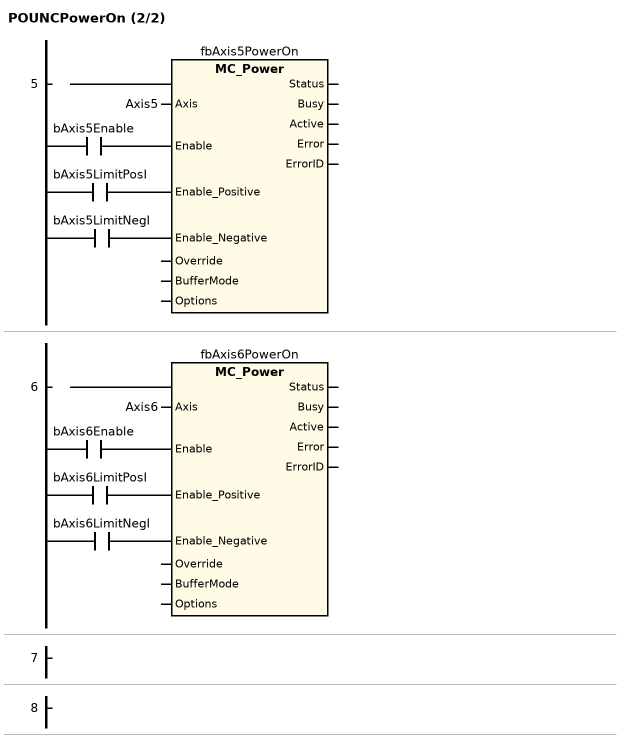
// NETWORK 5
fbAxis5PowerOn(
    Axis := Axis5,
    Enable := bAxis5Enable,
    Enable_Positive := bAxis5LimitPosI,
    Enable_Negative := bAxis5LimitNegI); // MC_Power

// NETWORK 6
fbAxis6PowerOn(
    Axis := Axis6,
    Enable := bAxis6Enable,
    Enable_Positive := bAxis6LimitPosI,
    Enable_Negative := bAxis6LimitNegI); // MC_Power

// NETWORK 7

// NETWORK 8

END_PROGRAM

// ---- POUs/POU_AxisJogCtrl.TcPOU
PROGRAM POU_AxisJogCtrl
VAR
	fb_Axis1Jog: MC_Jog;
	fb_Axis2Jog: MC_Jog;
END_VAR

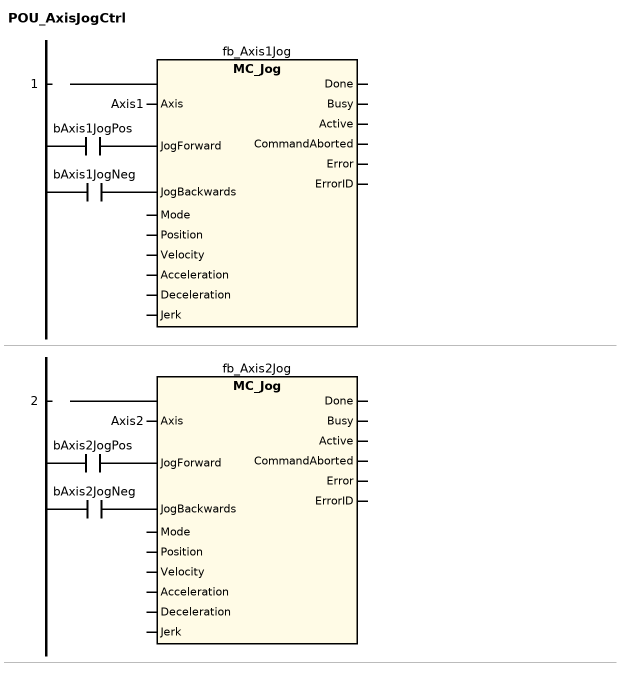
// NETWORK 1
fb_Axis1Jog(Axis := Axis1, JogForward := bAxis1JogPos, JogBackwards := bAxis1JogNeg); // MC_Jog

// NETWORK 2
fb_Axis2Jog(Axis := Axis2, JogForward := bAxis2JogPos, JogBackwards := bAxis2JogNeg); // MC_Jog

END_PROGRAM

// ---- POUs/POU_AxisMoveAbs.TcPOU
PROGRAM POU_AxisMoveAbs
VAR
	fbAxis1MoveAbs:MC_MoveAbsolute;
	fbAxis1MoveAbs2:MC_MoveAbsolute;
	fbAxis2MoveAbs:MC_MoveAbsolute;
	fbAxis2MoveAbs2:MC_MoveAbsolute;
	fbAxis3MoveAbs:MC_MoveAbsolute;
	fbAxis3MoveAbs2:MC_MoveAbsolute;
	fbAxis4MoveAbs:MC_MoveAbsolute;
	fbAxis4MoveAbs2:MC_MoveAbsolute;
	fbAxis5MoveAbs:MC_MoveAbsolute;
	fbAxis5MoveAbs2:MC_MoveAbsolute;
	fbAxis6MoveAbs:MC_MoveAbsolute;
	fbAxis6MoveAbs2:MC_MoveAbsolute;
END_VAR

//Set Vertical Velocities
rAxisVelV:=0.5;
rAxis2Vel:=rAxisVelV;
rAxis4Vel:=rAxisVelV;
rAxis6Vel:=rAxisVelV;
//Set Horizontal Velocities
rAxisVelH:=1;
rAxis1Vel:=rAxisVelH;
rAxis3Vel:=rAxisVelH;
rAxis5Vel:=rAxisVelH;
//Create Each Move and Seccondary
fbAxis1MoveAbs(
	Axis:= Axis1, 
	Execute:= , 
	Position:=rAxis1Target , 
	Velocity:= rAxis1Vel, 
	Acceleration:= , 
	Deceleration:= , 
	Jerk:= , 
	BufferMode:=MC_BlendingLow , 
	Options:= , 
	Done=> , 
	Busy=> , 
	Active=> , 
	CommandAborted=> , 
	Error=> , 
	ErrorID=> );

fbAxis1MoveAbs2(
	Axis:= Axis1, 
	Execute:= , 
	Position:=rAxis1Target , 
	Velocity:=rAxis1Vel , 
	Acceleration:= , 
	Deceleration:= , 
	Jerk:= , 
	BufferMode:=MC_BlendingLow , 
	Options:= , 
	Done=> , 
	Busy=> , 
	Active=> , 
	CommandAborted=> , 
	Error=> , 
	ErrorID=> );
	
fbAxis2MoveAbs(
	Axis:= Axis2, 
	Execute:= , 
	Position:=rAxis2Target , 
	Velocity:= rAxis2Vel, 
	Acceleration:= , 
	Deceleration:= , 
	Jerk:= , 
	BufferMode:= MC_BlendingLow, 
	Options:= , 
	Done=> , 
	Busy=> , 
	Active=> , 
	CommandAborted=> , 
	Error=> , 
	ErrorID=> );
	
fbAxis2MoveAbs2(
	Axis:= Axis2, 
	Execute:= , 
	Position:=rAxis2Target , 
	Velocity:= rAxis2Vel, 
	Acceleration:= , 
	Deceleration:= , 
	Jerk:= , 
	BufferMode:=MC_BlendingLow , 
	Options:= , 
	Done=> , 
	Busy=> , 
	Active=> , 
	CommandAborted=> , 
	Error=> , 
	ErrorID=> );

fbAxis3MoveAbs(
	Axis:= Axis3, 
	Execute:= , 
	Position:=rAxis3Target , 
	Velocity:= rAxis3Vel, 
	Acceleration:= , 
	Deceleration:= , 
	Jerk:= , 
	BufferMode:=MC_BlendingLow , 
	Options:= , 
	Done=> , 
	Busy=> , 
	Active=> , 
	CommandAborted=> , 
	Error=> , 
	ErrorID=> );
	
fbAxis3MoveAbs2(
	Axis:= Axis3, 
	Execute:= , 
	Position:=rAxis3Target , 
	Velocity:= rAxis3Vel, 
	Acceleration:= , 
	Deceleration:= , 
	Jerk:= , 
	BufferMode:=MC_BlendingLow , 
	Options:= , 
	Done=> , 
	Busy=> , 
	Active=> , 
	CommandAborted=> , 
	Error=> , 
	ErrorID=> );
	
fbAxis4MoveAbs(
	Axis:= Axis4, 
	Execute:= , 
	Position:=rAxis4Target , 
	Velocity:= rAxis4Vel, 
	Acceleration:= , 
	Deceleration:= , 
	Jerk:= , 
	BufferMode:=MC_BlendingLow , 
	Options:= , 
	Done=> , 
	Busy=> , 
	Active=> , 
	CommandAborted=> , 
	Error=> , 
	ErrorID=> );
	
fbAxis4MoveAbs2(
	Axis:= Axis4, 
	Execute:= , 
	Position:=rAxis4Target , 
	Velocity:= rAxis4Vel, 
	Acceleration:= , 
	Deceleration:= , 
	Jerk:= , 
	BufferMode:=MC_BlendingLow , 
	Options:= , 
	Done=> , 
	Busy=> , 
	Active=> , 
	CommandAborted=> , 
	Error=> , 
	ErrorID=> );
	
fbAxis5MoveAbs(
	Axis:= Axis5, 
	Execute:= , 
	Position:=rAxis5Target , 
	Velocity:=rAxis5Vel , 
	Acceleration:= , 
	Deceleration:= , 
	Jerk:= , 
	BufferMode:=MC_BlendingLow , 
	Options:= , 
	Done=> , 
	Busy=> , 
	Active=> , 
	CommandAborted=> , 
	Error=> , 
	ErrorID=> );
	
fbAxis5MoveAbs2(
	Axis:= Axis5, 
	Execute:= , 
	Position:=rAxis5Target , 
	Velocity:= rAxis5Vel, 
	Acceleration:= , 
	Deceleration:= , 
	Jerk:= , 
	BufferMode:=MC_BlendingLow , 
	Options:= , 
	Done=> , 
	Busy=> , 
	Active=> , 
	CommandAborted=> , 
	Error=> , 
	ErrorID=> );
	
fbAxis6MoveAbs(
	Axis:= Axis6, 
	Execute:= , 
	Position:=rAxis6Target , 
	Velocity:= rAxis6Vel, 
	Acceleration:= , 
	Deceleration:= , 
	Jerk:= , 
	BufferMode:=MC_BlendingLow , 
	Options:= , 
	Done=> , 
	Busy=> , 
	Active=> , 
	CommandAborted=> , 
	Error=> , 
	ErrorID=> );
	
fbAxis6MoveAbs2(
	Axis:= Axis6, 
	Execute:= , 
	Position:=rAxis6Target , 
	Velocity:= rAxis6Vel, 
	Acceleration:= , 
	Deceleration:= , 
	Jerk:= , 
	BufferMode:= MC_BlendingLow, 
	Options:= , 
	Done=> , 
	Busy=> , 
	Active=> , 
	CommandAborted=> , 
	Error=> , 
	ErrorID=> );
	


	IF bAxis1Enable	THEN
		IF bAxis1MoveABS THEN
			IF fbAxis1MoveAbs.Busy THEN
				IF fbAxis1MoveAbs2.Busy	THEN
					;
				ELSE
					fbAxis1MoveAbs2.Execute:=TRUE;
					bAxis1MoveAbs:=FALSE;
				END_IF
			ELSE
				fbAxis1MoveAbs.Execute:=TRUE;
				bAxis1MoveAbs:=FALSE;
			END_IF
		ELSIF fbAxis1MoveAbs.Done THEN
			bAxis1MoveAbs:=FALSE;
			fbAxis1MoveAbs.Execute:=FALSE;
		ELSIF fbAxis1MoveAbs2.Done THEN
			bAxis1MoveAbs:=FALSE;
			fbAxis1MoveAbs2.Execute:=FALSE;
		END_IF
	ELSE 
		fbAxis1MoveAbs2.Execute:=FALSE;
		fbAxis1MoveAbs.Execute:=FALSE;
	END_IF
	
	IF bAxis2Enable THEN
		IF bAxis2MoveABS THEN
			IF fbAxis2MoveAbs.Busy THEN
				IF fbAxis2MoveAbs2.Busy THEN
				;
				ELSE	
					fbAxis2MoveAbs2.Execute:=TRUE;
					bAxis2MoveAbs:=FALSE;
				END_IF
			ELSE
				fbAxis2MoveAbs.Execute:=TRUE;
				bAxis2MoveAbs:=FALSE;
			END_IF
		ELSIF fbAxis2MoveAbs.Done THEN
			bAxis2MoveAbs:=FALSE;
			fbAxis2MoveAbs.Execute:=FALSE;
		ELSIF fbAxis2MoveAbs2.Done THEN
			bAxis2MoveAbs:=FALSE;
			fbAxis2MoveAbs2.Execute:=FALSE;
		END_IF
	ELSE 
		fbAxis2MoveAbs2.Execute:=FALSE;
		fbAxis2MoveAbs.Execute:=FALSE;
	END_IF
	
	IF bAxis3Enable THEN
		IF bAxis3MoveABS THEN
			IF fbAxis3MoveAbs.Busy THEN
				IF fbAxis3MoveAbs2.Busy THEN
					;
				ELSE
					fbAxis3MoveAbs2.Execute:=TRUE;
					bAxis3MoveAbs:=FALSE;
				END_IF
			ELSE
				fbAxis3MoveAbs.Execute:=TRUE;
				bAxis3MoveAbs:=FALSE;
			END_IF
		ELSIF fbAxis3MoveAbs.Done THEN
			bAxis3MoveAbs:=FALSE;
			fbAxis3MoveAbs.Execute:=FALSE;
		ELSIF fbAxis3MoveAbs2.Done THEN
			bAxis3MoveAbs:=FALSE;
			fbAxis3MoveAbs2.Execute:=FALSE;
		END_IF
	ELSE 
		fbAxis3MoveAbs2.Execute:=FALSE;
		fbAxis3MoveAbs.Execute:=FALSE;
	END_IF
	
	IF bAxis4Enable THEN
		IF bAxis4MoveABS THEN
			IF fbAxis4MoveAbs.Busy THEN
				IF fbAxis4MoveAbs2.Busy THEN
					;
				ELSE
					fbAxis4MoveAbs2.Execute:=TRUE;
					bAxis4MoveAbs:=FALSE;
				END_IF
			ELSE
				fbAxis4MoveAbs.Execute:=TRUE;
				bAxis4MoveAbs:=FALSE;
			END_IF
		ELSIF fbAxis4MoveAbs.Done THEN
			bAxis4MoveAbs:=FALSE;
			fbAxis4MoveAbs.Execute:=FALSE;
		ELSIF fbAxis4MoveAbs2.Done THEN
			bAxis4MoveAbs:=FALSE;
			fbAxis4MoveAbs2.Execute:=FALSE;
			
		END_IF		
	ELSE 
		fbAxis4MoveAbs2.Execute:=FALSE;
		fbAxis4MoveAbs.Execute:=FALSE;
	END_IF
	
	IF bAxis5Enable THEN
		IF bAxis5MoveABS THEN
			IF fbAxis5MoveAbs.Busy THEN
				IF fbAxis5MoveAbs2.Busy THEN
					;
				ELSE
					fbAxis5MoveAbs2.Execute:=TRUE;
					bAxis5MoveAbs:=FALSE;
				END_IF
			ELSE
				fbAxis5MoveAbs.Execute:=TRUE;
				bAxis5MoveAbs:=FALSE;
			END_IF
		ELSIF fbAxis5MoveAbs.Done THEN
			bAxis5MoveAbs:=FALSE;
			fbAxis5MoveAbs.Execute:=FALSE;
		ELSIF fbAxis5MoveAbs2.Done THEN
			bAxis5MoveAbs:=FALSE;
			fbAxis5MoveAbs2.Execute:=FALSE;
		END_IF
	ELSE 
		fbAxis5MoveAbs2.Execute:=FALSE;
		fbAxis5MoveAbs.Execute:=FALSE;
	END_IF
	
	IF bAxis6Enable THEN
		IF bAxis6MoveABS THEN
			IF fbAxis6MoveAbs.Busy THEN
				IF fbAxis6MoveAbs2.Busy THEN
					;
				ELSE
					fbAxis6MoveAbs2.Execute:=TRUE;
					bAxis6MoveAbs:=FALSE;
				END_IF
			ELSE
				fbAxis6MoveAbs.Execute:=TRUE;
				bAxis6MoveAbs:=FALSE;
			END_IF
		ELSIF fbAxis6MoveAbs.Done THEN
			bAxis6MoveAbs:=FALSE;
			fbAxis6MoveAbs.Execute:=FALSE;
		ELSIF fbAxis6MoveAbs2.Done THEN
			bAxis6MoveAbs:=FALSE;
			fbAxis6MoveAbs2.Execute:=FALSE;
		ELSE 
			fbAxis6MoveAbs2.Execute:=FALSE;
			fbAxis6MoveAbs.Execute:=FALSE;
		END_IF
	ELSE 
		fbAxis6MoveAbs2.Execute:=FALSE;
		fbAxis6MoveAbs.Execute:=FALSE;
	END_IF

END_PROGRAM

// ---- POUs/POU_ClearAxesErrors.TcPOU
PROGRAM POU_ClearAxesErrors
VAR
	fbAxis1Reset:MC_Reset;
	fbAxis2Reset:MC_Reset;
	fbAxis3Reset:MC_Reset;
	fbAxis4Reset:MC_Reset;
	fbAxis5Reset:MC_Reset;
	fbAxis6Reset:MC_Reset;
	END_VAR


fbAxis1Reset(
	Axis:= Axis1, 
	Execute:=bReSetMotor , 
	Done=>bReset1Done , 
	Busy=> , 
	Error=> , 
	ErrorID=> );
	
fbAxis2Reset(
	Axis:= Axis2, 
	Execute:=bReSetMotor , 
	Done=>bReset2Done , 
	Busy=> , 
	Error=> , 
	ErrorID=> );
	
fbAxis3Reset(
	Axis:= Axis3, 
	Execute:=bReSetMotor , 
	Done=>bReset3Done , 
	Busy=> , 
	Error=> , 
	ErrorID=> );
	
fbAxis4Reset(
	Axis:= Axis4, 
	Execute:=bReSetMotor , 
	Done=>bReset4Done , 
	Busy=> , 
	Error=> , 
	ErrorID=> );
	
fbAxis5Reset(
	Axis:= Axis5, 
	Execute:=bReSetMotor , 
	Done=>bReset5Done , 
	Busy=> , 
	Error=> , 
	ErrorID=> );
	
fbAxis6Reset(
	Axis:= Axis6, 
	Execute:=bReSetMotor , 
	Done=>bReset6Done , 
	Busy=> , 
	Error=> , 
	ErrorID=> );

END_PROGRAM

// ---- POUs/POU_AbortMoves.TcPOU
PROGRAM POU_AbortMoves
VAR
	fbAxis1Halt:MC_Halt;
	fbAxis2Halt:MC_Halt;
	fbAxis3Halt:MC_Halt;
	fbAxis4Halt:MC_Halt;
	fbAxis5Halt:MC_Halt;
	fbAxis6Halt:MC_Halt;
	
END_VAR

fbAxis1Halt(
	Axis:= , 
	Execute:= , 
	Deceleration:= , 
	Jerk:= , 
	BufferMode:= , 
	Options:= , 
	Done=> , 
	Busy=> , 
	Active=> , 
	CommandAborted=> , 
	Error=> , 
	ErrorID=> );
	
fbAxis2Halt(
	Axis:= , 
	Execute:= , 
	Deceleration:= , 
	Jerk:= , 
	BufferMode:= , 
	Options:= , 
	Done=> , 
	Busy=> , 
	Active=> , 
	CommandAborted=> , 
	Error=> , 
	ErrorID=> );
	
fbAxis3Halt(
	Axis:= , 
	Execute:= , 
	Deceleration:= , 
	Jerk:= , 
	BufferMode:= , 
	Options:= , 
	Done=> , 
	Busy=> , 
	Active=> , 
	CommandAborted=> , 
	Error=> , 
	ErrorID=> );
	
fbAxis4Halt(
	Axis:= , 
	Execute:= , 
	Deceleration:= , 
	Jerk:= , 
	BufferMode:= , 
	Options:= , 
	Done=> , 
	Busy=> , 
	Active=> , 
	CommandAborted=> , 
	Error=> , 
	ErrorID=> );
	
fbAxis5Halt(
	Axis:= , 
	Execute:= , 
	Deceleration:= , 
	Jerk:= , 
	BufferMode:= , 
	Options:= , 
	Done=> , 
	Busy=> , 
	Active=> , 
	CommandAborted=> , 
	Error=> , 
	ErrorID=> );
	
fbAxis6Halt(
	Axis:= , 
	Execute:= , 
	Deceleration:= , 
	Jerk:= , 
	BufferMode:= , 
	Options:= , 
	Done=> , 
	Busy=> , 
	Active=> , 
	CommandAborted=> , 
	Error=> , 
	ErrorID=> );

END_PROGRAM

// ---- POUs/POU_AxisClearError.TcPOU
PROGRAM POU_AxisClearError
VAR_INPUT
END_VAR
VAR
	fbAxis1Reset:MC_Reset;
	fbAxis2Reset:MC_Reset;
	fbAxis3Reset:MC_Reset;
	fbAxis4Reset:MC_Reset;
	fbAxis5Reset:MC_Reset;
	fbAxis6Reset:MC_Reset;
	
END_VAR

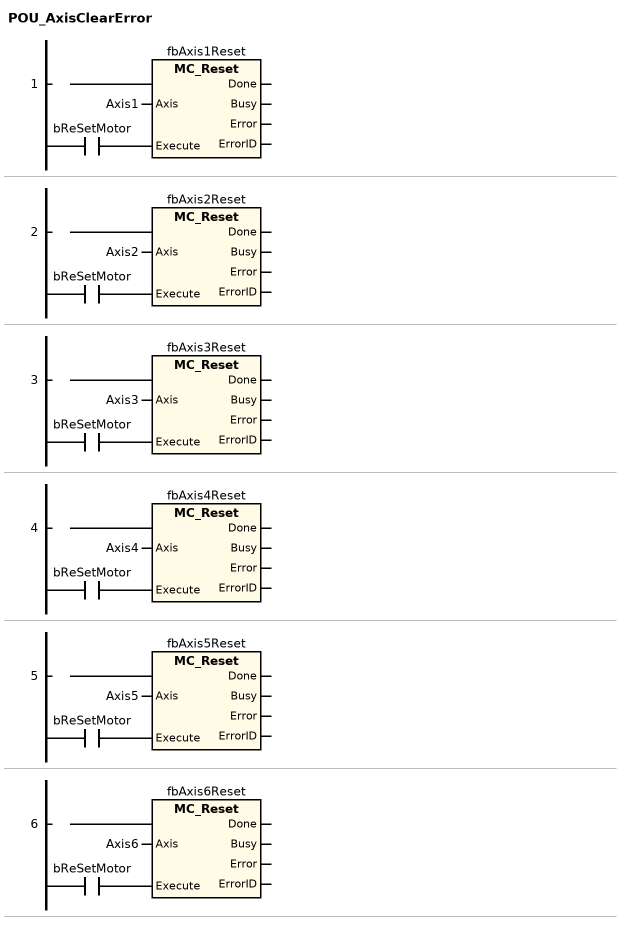
// NETWORK 1
fbAxis1Reset(Axis := Axis1, Execute := bReSetMotor); // MC_Reset

// NETWORK 2
fbAxis2Reset(Axis := Axis2, Execute := bReSetMotor); // MC_Reset

// NETWORK 3
fbAxis3Reset(Axis := Axis3, Execute := bReSetMotor); // MC_Reset

// NETWORK 4
fbAxis4Reset(Axis := Axis4, Execute := bReSetMotor); // MC_Reset

// NETWORK 5
fbAxis5Reset(Axis := Axis5, Execute := bReSetMotor); // MC_Reset

// NETWORK 6
fbAxis6Reset(Axis := Axis6, Execute := bReSetMotor); // MC_Reset

END_PROGRAM

// ---- POUs/POU_SetStatus.TcPOU
PROGRAM POU_SetStatus
VAR
END_VAR

END_PROGRAM

// ---- GlobalTextList.TcGTLO
TEXTLIST GlobalTextList
  76 = 'Clear error'
  18 = 'ENable'
  79 = 'Enable'
  614 = 'Jog Neg -'
  969 = 'Jog Plus +'
  194 = 'Jog Pos +'
  920 = 'Remote Control'
END_TEXTLIST

// ---- Visualizations/Visualization.TcVIS
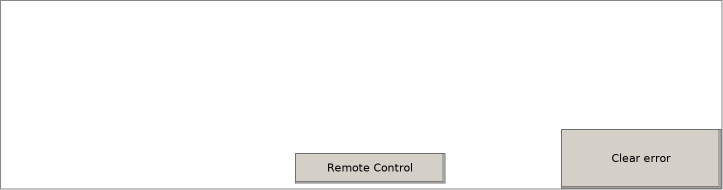
VISUALIZATION Visualization  // 723x190
    Button (295,153 150x30), "Remote Control"
        toggle bRemote
    Button (561,129 160x59), "Clear error"
END_VISUALIZATION
